PROGRAM P_Demo_FB_BARShadingCorrectionSouth
VAR
    fb : FB_BARShadingCorrectionSouth;                            // 被演示 FB 实例
    eDataSecurityType_in : E_HVACDataSecurityType ;
    stTimeAct_in : TIMESTRUCT ;
    lrAzimuth_in : LREAL := 0.0;
    lrElevation_in : LREAL := 0.0;
    arrFacadeElement_io : ARRAY[1..iColumnsPerFacade, 1..iRowsPerFacade] OF ST_BARFacadeElement ;
    arrShadingObject_io : ARRAY[1..iShadingObjects] OF ST_BARShadingObject ;
    lrFacadeOrientation_io : LREAL := 0.0;
    usiGroupID_io : USINT := 0;
    bGroupNotShaded_out : BOOL;
    bFacadeSunlit_out : BOOL;
    bError_out : BOOL;
    udiErrorId_out : UDINT;
END_VAR

// ============================================================================
// Tc2_HVAC.FB_BARShadingCorrectionSouth 演示程序
// ============================================================================
// 场景：把本 FB 实例化到一个 PLC 程序里，每周期单次调用；按需要把 VAR_INPUT 与
//       VAR_IN_OUT 接到工程信号；VAR_OUTPUT 写入对应监视变量。
// 价值：使用本 FB 比手写状态机 / 控制算法节省大量代码；与 Tc2_HVAC 体系内其它 FB
//       直接对接，命名 / 持久化 / 模式仲裁等约定一致。具体语义见 FB_BARShadingCorrectionSouth.md 主文档。
// 验证步骤：
//   1. 右键 PLC 项目下 POUs 文件夹 → Add → Existing Item → 选本 .TcPOU 文件
//   2. 引用 Tc2_HVAC（References → Add library）
//   3. 编译 → 登录 → 运行
//   4. 在线写各 *_in 输入信号触发 FB；在线 monitor *_out 引脚观察状态
// ============================================================================

fb(
    eDataSecurityType := eDataSecurityType_in,
    stTimeAct := stTimeAct_in,
    lrAzimuth := lrAzimuth_in,
    lrElevation := lrElevation_in,
    arrFacadeElement := arrFacadeElement_io,
    arrShadingObject := arrShadingObject_io,
    lrFacadeOrientation := lrFacadeOrientation_io,
    usiGroupID := usiGroupID_io,
    bGroupNotShaded => bGroupNotShaded_out,
    bFacadeSunlit => bFacadeSunlit_out,
    bError => bError_out,
    udiErrorId => udiErrorId_out
);

END_PROGRAM

(* stored: Version 1.1.0.1, ProductVersion 3.1.4024.5
   POU P_Demo_FB_BARShadingCorrectionSouth: Id {be4c82e8-0fe2-5b3e-a5ff-2390680ef276}, SpecialFunc None *)
